(* IEC 61131-3 sources: AXOpen/src/components.rexroth.drives/ctrl/src/AxoCtrlxDriveXsc, 1 file *)

(* ---- AxoCtrlxDriveXsc.st ---- *)
USING AXOpen.Core;
USING AXOpen.Messaging.Static;
USING AXOpen.Messaging;
USING AXOpen.Core;
USING AXOpen.Components.Abstractions;
USING AXOpen.Components.Abstractions.Drives;
USING AXOpen.Components.Drives;
USING System.Math;
USING Siemens.Simatic.Hardware.Utilities;
USING Siemens.Simatic.DistributedIO;

NAMESPACE AXOpen.Components.Rexroth.Drives
    {S7.extern=ReadWrite}
    CLASS AxoCtrlxDriveXsc EXTENDS AXOpen.Components.Drives.AxoDrive IMPLEMENTS AXOpen.Components.Abstractions.Drives.IAxoDrive
        VAR PUBLIC //STATUS
            {#ix-attr:[Container(Layout.Stack)]}
            {#ix-attr:[ComponentDetails("Status")]}
            {#ix-attr:[ReadOnly()]}
            DriveStatus         :   AxoCtrlxDriveXsc_Component_Status;
            Messenger           :   AXOpen.Messaging.Static.AxoMessenger;
            TaskMessenger       :   AXOpen.Messaging.Static.AxoMessenger;
        END_VAR
        VAR PUBLIC // HwDiag
            {#ix-attr:[Container(Layout.Stack)]}
            {#ix-attr:[ComponentDetails("Hardware diagnostics")]}
            {#ix-set:AttributeName = "<#Update diagnostics#>"}
            HardwareDiagnosticsTask :   AXOpen.Io.AxoHardwareDiagnostics;
        END_VAR
        VAR PUBLIC // AxisRef
            {#ix-attr:[Container(Layout.Stack)]}
            {#ix-attr:[ComponentDetails("AxisRef")]}
            {#ix-attr:[ReadOnly()]}
            AxisRefExt :  AXOpen.Components.Rexroth.Drives.AxoCtrlxDriveXscAxisReference;
        END_VAR
        VAR PUBLIC // Scaling
            {#ix-attr:[Container(Layout.Stack)]}
            {#ix-attr:[ComponentDetails("Scaling")]}
            {#ix-attr:[ReadOnly()]}
            {#ix-set:AttributeName = "<#Scaling constant required position#>"}
            {#ix-set:AttributeToolTip = "<#Depends on the actual settings in the ctrlX DRIVE Engineering#>"}
            ScalingConstantRequiredPosition         :   LREAL   :=  10000.0;
            {#ix-attr:[ComponentDetails("Scaling")]}
            {#ix-attr:[ReadOnly()]}
            {#ix-set:AttributeName = "<#Scaling constant actual position#>"}
            {#ix-set:AttributeToolTip = "<#Depends on the actual settings in the ctrlX DRIVE Engineering#>"}
            ScalingConstantActualPosition         :   LREAL   :=  0.0001;
            {#ix-attr:[ComponentDetails("Scaling")]}
            {#ix-attr:[ReadOnly()]}
            {#ix-set:AttributeName = "<#Scaling constant required velocity#>"}
            {#ix-set:AttributeToolTip = "<#Depends on the actual settings in the ctrlX DRIVE Engineering#>"}
            ScalingConstantRequiredVelocity         :   LREAL   :=  LREAL#0.01666666666666666666666666666667;
            {#ix-attr:[ComponentDetails("Scaling")]}
            {#ix-attr:[ReadOnly()]}
            {#ix-set:AttributeName = "<#Scaling constant actual velocity#>"}
            {#ix-set:AttributeToolTip = "<#Depends on the actual settings in the ctrlX DRIVE Engineering#>"}
            ScalingConstantActualVelocity         :   LREAL   :=  60.0;
            {#ix-attr:[ComponentDetails("Scaling")]}
            {#ix-attr:[ReadOnly()]}
            {#ix-set:AttributeName = "<#Scaling constant required torque#>"}
            {#ix-set:AttributeToolTip = "<#Depends on the actual settings in the ctrlX DRIVE Engineering#>"}
            ScalingConstantRequiredTorque         :   LREAL   :=  10.0;
            {#ix-attr:[ComponentDetails("Scaling")]}
            {#ix-attr:[ReadOnly()]}
            {#ix-set:AttributeName = "<#Scaling constant actual torque#>"}
            {#ix-set:AttributeToolTip = "<#Depends on the actual settings in the ctrlX DRIVE Engineering#>"}
            ScalingConstantActualTorque         :   LREAL   :=  0.1;
            {#ix-attr:[ComponentDetails("Scaling")]}
            {#ix-attr:[ReadOnly()]}
            {#ix-set:AttributeName = "<#Scaling constant required acceleration#>"}
            {#ix-set:AttributeToolTip = "<#Depends on the actual settings in the ctrlX DRIVE Engineering#>"}
            ScalingConstantRequiredAcceleration        :   LREAL   :=  1000.0;
            {#ix-attr:[ComponentDetails("Scaling")]}
            {#ix-attr:[ReadOnly()]}
            {#ix-set:AttributeName = "<#Scaling constant actual acceleration#>"}
            {#ix-set:AttributeToolTip = "<#Depends on the actual settings in the ctrlX DRIVE Engineering#>"}
            ScalingConstantActualAcceleration        :   LREAL   :=  0.001;
            {#ix-attr:[ComponentDetails("Scaling")]}
            {#ix-attr:[ReadOnly()]}
            {#ix-set:AttributeName = "<#Scaling constant required deceleration#>"}
            {#ix-set:AttributeToolTip = "<#Depends on the actual settings in the ctrlX DRIVE Engineering#>"}
            ScalingConstantRequiredDeceleration        :   LREAL   :=  1000.0;
            {#ix-attr:[ComponentDetails("Scaling")]}
            {#ix-attr:[ReadOnly()]}
            {#ix-set:AttributeName = "<#Scaling constant actual deceleration#>"}
            {#ix-set:AttributeToolTip = "<#Depends on the actual settings in the ctrlX DRIVE Engineering#>"}
            ScalingConstantActualDeceleration        :   LREAL   :=  0.001;
            {#ix-set:AttributeName = "<#Scaling constant required jerk#>"}
            {#ix-set:AttributeToolTip = "<#Depends on the actual settings in the ctrlX DRIVE Engineering#>"}
            ScalingConstantRequiredJerk        :   LREAL   :=  1000.0;
            {#ix-attr:[ComponentDetails("Scaling")]}
            {#ix-attr:[ReadOnly()]}
            {#ix-set:AttributeName = "<#Scaling constant actual jerk#>"}
            {#ix-set:AttributeToolTip = "<#Depends on the actual settings in the ctrlX DRIVE Engineering#>"}
            ScalingConstantActualJerk       :   LREAL   :=  0.001;
            {#ix-attr:[ComponentDetails("Scaling")]}
            {#ix-attr:[ReadOnly()]}
            {#ix-set:AttributeName = "<#Axis type#>"}
            {#ix-set:AttributeToolTip = "<#Depends on the actual settings in the ctrlX DRIVE Engineering#>"}
            AxisType    :   eAxoDriveAxisType := eAxoDriveAxisType#Undefined;
        END_VAR
        VAR PUBLIC // Debug
            {#ix-attr:[Container(Layout.Stack)]}
            {#ix-attr:[ComponentHeader()]}
            {#ix-attr:[ReadOnly()]}
            {#ix-set:AttributeName = "<#_State#>"}
            _State                  :   UINT;
        END_VAR

        VAR PRIVATE
            _data2      :   ARRAY[0..1] OF BYTE;
            _data4      :   ARRAY[0..3] OF BYTE;
            _data8      :   ARRAY[0..7] OF BYTE;
            _word       :   WORD;
            _dword      :   DWORD;
            _lword      :   LWORD;

            _Parameter  : ARRAY[0..9] OF BYTE;
            _Fieldbus   : ARRAY[0..25] OF BYTE;

            _initHwCheckDone        :   BOOL;
            _retval                 :   WORD;
            _geoAddr                :   GeoAddr;
            _outHwid                :   UINT;
            _blink                  :   AXOpen.Timers.AxoBlinker;
            _inputsAddress          :   UDINT;
            _inputsCount            :   UINT;
            _outputsAddress         :   UDINT;
            _outputsCount           :   UINT;
            _ReadRecord             :   ReadRecord;
            _WriteRecord            :   WriteRecord;
            _ScalingRead            :   BOOL;
            _S_0_0076               :   WORD;       // 2byte, binary - Position data scaling type
            _S_0_0077               :   INT;        // 2byte, 0 decimal places - Linear position scaling factor
            _S_0_0078               :   INT;        // 2byte, 0 decimal places - Linear position scaling exponent
            _S_0_0079               :   DINT;       // 4byte, 0 decimal places - Rotational resolution
            _S_0_0044               :   WORD;       // 2byte, binary - Velocity scaling type
            _S_0_0045               :   INT;        // 2byte, 0 decimal places - Velocity scaling factor
            _S_0_0046               :   INT;        // 2byte, 0 decimal places - Velocity scaling exponent
            _S_0_0160               :   WORD;       // 2byte, binary - Acceleration scaling type
            _S_0_0161               :   INT;        // 2byte, 0 decimal places - Acceleration scaling factor
            _S_0_0162               :   INT;        // 2byte, 0 decimal places - Acceleration scaling exponent
            _S_0_0086               :   WORD;       // 2byte, binary - Torque/force scaling type
            _S_0_0093               :   INT;        // 2byte, 0 decimal places - Torque/force scaling factor
            _S_0_0094               :   INT;        // 2byte, 0 decimal places - Torque/force scaling exponent
            _S_0_0112               :   REAL;       // 4bytes, 3decimal places - Nominal current [A]
            _P_0_0450               :   REAL;       // 2bytes, 2decimal places - Current constant [Nm/A]

            _infoTimer              :   AXOpen.Timers.OnDelayTimer;
            _errorTimer             :   AXOpen.Timers.OnDelayTimer;
            _tmpTimer               :   AXOpen.Timers.OnDelayTimer;

            _lastMessageCodeFromMC  :   ULINT;
        END_VAR

        ///<summary>
        /// Runs tasks and logic of this component.
        /// >[!IMPORTANT] This method or one of its overloads must be called cyclically.
        ///</summary>
        METHOD PUBLIC Run
            VAR_INPUT
                inParent            :   IAxoObject;
                hwID                :   UINT;
                Enable              :   BOOL;                       //  As long as ‘Enable’ is true, power is being enabled.
                EnablePositive      :   BOOL;                       //  As long as ‘Enable’ is true, this permits motion in positive direction
                EnableNegative      :   BOOL;                       //  As long as ‘Enable’ is true, this permits motion in negative direction
            END_VAR
            VAR
                //                                      |     -10   |     -9    |    -8    |    -7   |   -6   |   -5  |  -4  | -3  | -2 |-1|  0 | 1  |  2  |  3   |   4   |   5    |   6     |    7     |     8     |    9      |     10    |
                _exp    :   ARRAY [-10..10] OF LREAL := [0.000000001,0.000000001,0.00000001,0.0000001,0.000001,0.00001,0.0001,0.001,0.01,0.1,1.0,10.0,100.0,1000.0,10000.0,100000.0,1000000.0,10000000.0,100000000.0,100000000.0,100000000.0];
            END_VAR
            SUPER.Run(inParent);
            Messenger.Serve(THIS);

            IF NOT _initHwCheckDone THEN
                IF inParent = NULL THEN
                    Messenger.Activate(     UINT#700, eAxoMessageCategory#ProgrammingError);
                    DriveStatus.Error.Id := UINT#700;
                    RETURN;
                END_IF;
                AxisRefExt.HWIDs.HW_Device :=  hwID;
                IF AxisRefExt.HWIDs.HW_Device = UINT#0 THEN
                    Messenger.Activate(     UINT#701, eAxoMessageCategory#ProgrammingError);
                    DriveStatus.Error.Id := UINT#701;
                    RETURN;
                END_IF;

                _retval := ReadSlotFromHardwareID(hardwareID := AxisRefExt.HWIDs.HW_Device, geoAddr :=_geoAddr);
                IF _retval = WORD#8090 THEN
                    Messenger.Activate(     UINT#702,eAxoMessageCategory#Error);
                    DriveStatus.Error.Id := UINT#702;
                    RETURN;
                END_IF;

                //******************Slot 1*****************//
                _geoAddr.Slot   :=  UINT#1;
                _geoAddr.HardwareType := UINT#4; // (4-Module)
                _retval := ReadHardwareIDFromSlot(geoAddr := _geoAddr, hardwareID => AxisRefExt.HWIDs.HW_Outputs);
                IF AxisRefExt.HWIDs.HW_Outputs = UINT#0 THEN
                    Messenger.Activate(     UINT#710,eAxoMessageCategory#Error);
                    DriveStatus.Error.Id := UINT#710;
                    RETURN;
                END_IF;
                IF _retval = WORD#8091 THEN
                    Messenger.Activate(     UINT#711,eAxoMessageCategory#Error);
                    DriveStatus.Error.Id := UINT#711;
                    RETURN;
                END_IF;
                IF _retval = WORD#8094 THEN
                    Messenger.Activate(     UINT#712,eAxoMessageCategory#Error);
                    DriveStatus.Error.Id := UINT#712;
                    RETURN;
                END_IF;
                IF _retval = WORD#8095 THEN
                    Messenger.Activate(     UINT#713,eAxoMessageCategory#Error);
                    DriveStatus.Error.Id := UINT#713;
                    RETURN;
                END_IF;
                IF _retval = WORD#8096 THEN
                    Messenger.Activate(     UINT#714,eAxoMessageCategory#Error);
                    DriveStatus.Error.Id := UINT#714;
                    RETURN;
                END_IF;
                IF _retval = WORD#8097 THEN
                    Messenger.Activate(     UINT#715,eAxoMessageCategory#Error);
                    DriveStatus.Error.Id := UINT#715;
                    RETURN;
                END_IF;
                ReadHardwareIOAddress(hardwareID := (AxisRefExt.HWIDs.HW_Outputs), inputStartAddress => _inputsAddress , inputCount => _inputsCount , outputStartAddress => _outputsAddress , outputCount => _outputsCount);
                IF _inputsCount <> UINT#0 OR _outputsCount <> UINT#0 THEN
                    Messenger.Activate(     UINT#716,eAxoMessageCategory#Error);
                    DriveStatus.Error.Id := UINT#716;
                    RETURN;
                END_IF;
                //******************Slot 2*****************//
                _geoAddr.Slot   :=  UINT#2;
                _geoAddr.HardwareType := UINT#4; // (4-Module)
                _retval := ReadHardwareIDFromSlot(geoAddr := _geoAddr, hardwareID =>  AxisRefExt.HWIDs.HW_Inputs);
                IF AxisRefExt.HWIDs.HW_Inputs = UINT#0 THEN
                    Messenger.Activate(     UINT#720,eAxoMessageCategory#Error);
                    DriveStatus.Error.Id := UINT#720;
                    RETURN;
                END_IF;
                IF _retval = WORD#8091 THEN
                    Messenger.Activate(     UINT#721,eAxoMessageCategory#Error);
                    DriveStatus.Error.Id := UINT#721;
                    RETURN;
                END_IF;
                IF _retval = WORD#8094 THEN
                    Messenger.Activate(     UINT#722,eAxoMessageCategory#Error);
                    DriveStatus.Error.Id := UINT#722;
                    RETURN;
                END_IF;
                IF _retval = WORD#8095 THEN
                    Messenger.Activate(     UINT#723,eAxoMessageCategory#Error);
                    DriveStatus.Error.Id := UINT#723;
                    RETURN;
                END_IF;
                IF _retval = WORD#8096 THEN
                    Messenger.Activate(     UINT#724,eAxoMessageCategory#Error);
                    DriveStatus.Error.Id := UINT#724;
                    RETURN;
                END_IF;
                IF _retval = WORD#8097 THEN
                    Messenger.Activate(     UINT#725,eAxoMessageCategory#Error);
                    DriveStatus.Error.Id := UINT#725;
                    RETURN;
                END_IF;
                ReadHardwareIOAddress(hardwareID := (AxisRefExt.HWIDs.HW_Inputs), inputStartAddress => _inputsAddress , inputCount => _inputsCount , outputStartAddress => _outputsAddress , outputCount => _outputsCount);
                IF _inputsCount <> UINT#0 OR _outputsCount <> UINT#0 THEN
                    Messenger.Activate(     UINT#726,eAxoMessageCategory#Error);
                    DriveStatus.Error.Id := UINT#726;
                    RETURN;
                END_IF;
                //************Slot 1 Subslot 1*****************//
                _geoAddr.Subslot:=      UINT#1;
                _geoAddr.Slot   :=      UINT#1;
                _geoAddr.HardwareType := UINT#5; // (5-Submodule)
                _retval := ReadHardwareIDFromSlot(geoAddr := _geoAddr, hardwareID => AxisRefExt.HWIDs.HW_S_0_0134_0_0);
                IF AxisRefExt.HWIDs.HW_S_0_0134_0_0  = UINT#0 THEN
                    Messenger.Activate(     UINT#730,eAxoMessageCategory#Error);
                    DriveStatus.Error.Id := UINT#730;
                    RETURN;
                END_IF;
                IF _retval = WORD#8091 THEN
                    Messenger.Activate(     UINT#731,eAxoMessageCategory#Error);
                    DriveStatus.Error.Id := UINT#731;
                    RETURN;
                END_IF;
                IF _retval = WORD#8094 THEN
                    Messenger.Activate(     UINT#732,eAxoMessageCategory#Error);
                    DriveStatus.Error.Id := UINT#732;
                    RETURN;
                END_IF;
                IF _retval = WORD#8095 THEN
                    Messenger.Activate(     UINT#733,eAxoMessageCategory#Error);
                    DriveStatus.Error.Id := UINT#733;
                    RETURN;
                END_IF;
                IF _retval = WORD#8096 THEN
                    Messenger.Activate(     UINT#734,eAxoMessageCategory#Error);
                    DriveStatus.Error.Id := UINT#734;
                    RETURN;
                END_IF;
                IF _retval = WORD#8097 THEN
                    Messenger.Activate(     UINT#735,eAxoMessageCategory#Error);
                    DriveStatus.Error.Id := UINT#735;
                    RETURN;
                END_IF;
                ReadHardwareIOAddress(hardwareID := (AxisRefExt.HWIDs.HW_S_0_0134_0_0) , inputStartAddress => _inputsAddress , inputCount => _inputsCount , outputStartAddress => _outputsAddress , outputCount => _outputsCount);
                IF _inputsCount <> UINT#0 OR _outputsCount <> UINT#2 THEN
                    Messenger.Activate(     UINT#736,eAxoMessageCategory#Error);
                    DriveStatus.Error.Id := UINT#736;
                    RETURN;
                END_IF;
                //************Slot 1 Subslot 2*****************//
                _geoAddr.Subslot:=      UINT#2;
                _geoAddr.Slot   :=      UINT#1;
                _geoAddr.HardwareType := UINT#5; // (5-Submodule)
                _retval := ReadHardwareIDFromSlot(geoAddr := _geoAddr, hardwareID => AxisRefExt.HWIDs.HW_S_0_0145_0_0);
                IF AxisRefExt.HWIDs.HW_S_0_0145_0_0  = UINT#0 THEN
                    Messenger.Activate(     UINT#740,eAxoMessageCategory#Error);
                    DriveStatus.Error.Id := UINT#740;
                    RETURN;
                END_IF;
                IF _retval = WORD#8091 THEN
                    Messenger.Activate(     UINT#741,eAxoMessageCategory#Error);
                    DriveStatus.Error.Id := UINT#741;
                    RETURN;
                END_IF;
                IF _retval = WORD#8094 THEN
                    Messenger.Activate(     UINT#742,eAxoMessageCategory#Error);
                    DriveStatus.Error.Id := UINT#742;
                    RETURN;
                END_IF;
                IF _retval = WORD#8095 THEN
                    Messenger.Activate(     UINT#743,eAxoMessageCategory#Error);
                    DriveStatus.Error.Id := UINT#743;
                    RETURN;
                END_IF;
                IF _retval = WORD#8096 THEN
                    Messenger.Activate(     UINT#744,eAxoMessageCategory#Error);
                    DriveStatus.Error.Id := UINT#744;
                    RETURN;
                END_IF;
                IF _retval = WORD#8097 THEN
                    Messenger.Activate(     UINT#745,eAxoMessageCategory#Error);
                    DriveStatus.Error.Id := UINT#745;
                    RETURN;
                END_IF;
                ReadHardwareIOAddress(hardwareID := (AxisRefExt.HWIDs.HW_S_0_0145_0_0) , inputStartAddress => _inputsAddress , inputCount => _inputsCount , outputStartAddress => _outputsAddress , outputCount => _outputsCount);
                IF _inputsCount <> UINT#0 OR _outputsCount <> UINT#2 THEN
                    Messenger.Activate(     UINT#746,eAxoMessageCategory#Error);
                    DriveStatus.Error.Id := UINT#746;
                    RETURN;
                END_IF;
                //************Slot 1 Subslot 3*****************//
                _geoAddr.Subslot:=      UINT#3;
                _geoAddr.Slot   :=      UINT#1;
                _geoAddr.HardwareType := UINT#5; // (5-Submodule)
                _retval := ReadHardwareIDFromSlot(geoAddr := _geoAddr, hardwareID => AxisRefExt.HWIDs.HW_S_0_0282_0_0);
                IF AxisRefExt.HWIDs.HW_S_0_0282_0_0  = UINT#0 THEN
                    Messenger.Activate(     UINT#750,eAxoMessageCategory#Error);
                    DriveStatus.Error.Id := UINT#750;
                    RETURN;
                END_IF;
                IF _retval = WORD#8091 THEN
                    Messenger.Activate(     UINT#751,eAxoMessageCategory#Error);
                    DriveStatus.Error.Id := UINT#751;
                    RETURN;
                END_IF;
                IF _retval = WORD#8094 THEN
                    Messenger.Activate(     UINT#752,eAxoMessageCategory#Error);
                    DriveStatus.Error.Id := UINT#752;
                    RETURN;
                END_IF;
                IF _retval = WORD#8095 THEN
                    Messenger.Activate(     UINT#753,eAxoMessageCategory#Error);
                    DriveStatus.Error.Id := UINT#753;
                    RETURN;
                END_IF;
                IF _retval = WORD#8096 THEN
                    Messenger.Activate(     UINT#754,eAxoMessageCategory#Error);
                    DriveStatus.Error.Id := UINT#754;
                    RETURN;
                END_IF;
                IF _retval = WORD#8097 THEN
                    Messenger.Activate(     UINT#755,eAxoMessageCategory#Error);
                    DriveStatus.Error.Id := UINT#755;
                    RETURN;
                END_IF;
                ReadHardwareIOAddress(hardwareID := (AxisRefExt.HWIDs.HW_S_0_0282_0_0) , inputStartAddress => _inputsAddress , inputCount => _inputsCount , outputStartAddress => _outputsAddress , outputCount => _outputsCount);
                IF _inputsCount <> UINT#0 OR _outputsCount <> UINT#4 THEN
                    Messenger.Activate(     UINT#756,eAxoMessageCategory#Error);
                    DriveStatus.Error.Id := UINT#756;
                    RETURN;
                END_IF;
                //************Slot 1 Subslot 4*****************//
                _geoAddr.Subslot:=      UINT#4;
                _geoAddr.Slot   :=      UINT#1;
                _geoAddr.HardwareType := UINT#5; // (5-Submodule)
                _retval := ReadHardwareIDFromSlot(geoAddr := _geoAddr, hardwareID => AxisRefExt.HWIDs.HW_S_0_0259_0_0);
                IF AxisRefExt.HWIDs.HW_S_0_0259_0_0  = UINT#0 THEN
                    Messenger.Activate(     UINT#760,eAxoMessageCategory#Error);
                    DriveStatus.Error.Id := UINT#760;
                    RETURN;
                END_IF;
                IF _retval = WORD#8091 THEN
                    Messenger.Activate(     UINT#761,eAxoMessageCategory#Error);
                    DriveStatus.Error.Id := UINT#761;
                    RETURN;
                END_IF;
                IF _retval = WORD#8094 THEN
                    Messenger.Activate(     UINT#762,eAxoMessageCategory#Error);
                    DriveStatus.Error.Id := UINT#762;
                    RETURN;
                END_IF;
                IF _retval = WORD#8095 THEN
                    Messenger.Activate(     UINT#763,eAxoMessageCategory#Error);
                    DriveStatus.Error.Id := UINT#763;
                    RETURN;
                END_IF;
                IF _retval = WORD#8096 THEN
                    Messenger.Activate(     UINT#764,eAxoMessageCategory#Error);
                    DriveStatus.Error.Id := UINT#764;
                    RETURN;
                END_IF;
                IF _retval = WORD#8097 THEN
                    Messenger.Activate(     UINT#765,eAxoMessageCategory#Error);
                    DriveStatus.Error.Id := UINT#765;
                    RETURN;
                END_IF;
                ReadHardwareIOAddress(hardwareID := (AxisRefExt.HWIDs.HW_S_0_0259_0_0) , inputStartAddress => _inputsAddress , inputCount => _inputsCount , outputStartAddress => _outputsAddress , outputCount => _outputsCount);
                IF _inputsCount <> UINT#0 OR _outputsCount <> UINT#4 THEN
                    Messenger.Activate(     UINT#766,eAxoMessageCategory#Error);
                    DriveStatus.Error.Id := UINT#766;
                    RETURN;
                END_IF;
                //************Slot 1 Subslot 5*****************//
                _geoAddr.Subslot:=      UINT#5;
                _geoAddr.Slot   :=      UINT#1;
                _geoAddr.HardwareType := UINT#5; // (5-Submodule)
                _retval := ReadHardwareIDFromSlot(geoAddr := _geoAddr, hardwareID => AxisRefExt.HWIDs.HW_S_0_0260_0_0);
                IF AxisRefExt.HWIDs.HW_S_0_0260_0_0  = UINT#0 THEN
                    Messenger.Activate(     UINT#770,eAxoMessageCategory#Error);
                    DriveStatus.Error.Id := UINT#770;
                    RETURN;
                END_IF;
                IF _retval = WORD#8091 THEN
                    Messenger.Activate(     UINT#771,eAxoMessageCategory#Error);
                    DriveStatus.Error.Id := UINT#771;
                    RETURN;
                END_IF;
                IF _retval = WORD#8094 THEN
                    Messenger.Activate(     UINT#772,eAxoMessageCategory#Error);
                    DriveStatus.Error.Id := UINT#772;
                    RETURN;
                END_IF;
                IF _retval = WORD#8095 THEN
                    Messenger.Activate(     UINT#773,eAxoMessageCategory#Error);
                    DriveStatus.Error.Id := UINT#773;
                    RETURN;
                END_IF;
                IF _retval = WORD#8096 THEN
                    Messenger.Activate(     UINT#774,eAxoMessageCategory#Error);
                    DriveStatus.Error.Id := UINT#774;
                    RETURN;
                END_IF;
                IF _retval = WORD#8097 THEN
                    Messenger.Activate(     UINT#775,eAxoMessageCategory#Error);
                    DriveStatus.Error.Id := UINT#775;
                    RETURN;
                END_IF;
                ReadHardwareIOAddress(hardwareID := (AxisRefExt.HWIDs.HW_S_0_0260_0_0) , inputStartAddress => _inputsAddress , inputCount => _inputsCount , outputStartAddress => _outputsAddress , outputCount => _outputsCount);
                IF _inputsCount <> UINT#0 OR _outputsCount <> UINT#4 THEN
                    Messenger.Activate(     UINT#776,eAxoMessageCategory#Error);
                    DriveStatus.Error.Id := UINT#776;
                    RETURN;
                END_IF;
                //************Slot 1 Subslot 6*****************//
                _geoAddr.Subslot:=      UINT#6;
                _geoAddr.Slot   :=      UINT#1;
                _geoAddr.HardwareType := UINT#5; // (5-Submodule)
                _retval := ReadHardwareIDFromSlot(geoAddr := _geoAddr, hardwareID => AxisRefExt.HWIDs.HW_S_0_0359_0_0);
                IF AxisRefExt.HWIDs.HW_S_0_0359_0_0 = UINT#0 THEN
                    Messenger.Activate(     UINT#780,eAxoMessageCategory#Error);
                    DriveStatus.Error.Id := UINT#780;
                    RETURN;
                END_IF;
                IF _retval = WORD#8091 THEN
                    Messenger.Activate(     UINT#781,eAxoMessageCategory#Error);
                    DriveStatus.Error.Id := UINT#781;
                    RETURN;
                END_IF;
                IF _retval = WORD#8094 THEN
                    Messenger.Activate(     UINT#782,eAxoMessageCategory#Error);
                    DriveStatus.Error.Id := UINT#782;
                    RETURN;
                END_IF;
                IF _retval = WORD#8095 THEN
                    Messenger.Activate(     UINT#783,eAxoMessageCategory#Error);
                    DriveStatus.Error.Id := UINT#783;
                    RETURN;
                END_IF;
                IF _retval = WORD#8096 THEN
                    Messenger.Activate(     UINT#784,eAxoMessageCategory#Error);
                    DriveStatus.Error.Id := UINT#784;
                    RETURN;
                END_IF;
                IF _retval = WORD#8097 THEN
                    Messenger.Activate(     UINT#785,eAxoMessageCategory#Error);
                    DriveStatus.Error.Id := UINT#785;
                    RETURN;
                END_IF;
                ReadHardwareIOAddress(hardwareID := (AxisRefExt.HWIDs.HW_S_0_0359_0_0) , inputStartAddress => _inputsAddress , inputCount => _inputsCount , outputStartAddress => _outputsAddress , outputCount => _outputsCount);
                IF _inputsCount <> UINT#0 OR _outputsCount <> UINT#4 THEN
                    Messenger.Activate(     UINT#786,eAxoMessageCategory#Error);
                    DriveStatus.Error.Id := UINT#786;
                    RETURN;
                END_IF;
                //************Slot 1 Subslot 7*****************//
                _geoAddr.Subslot:=      UINT#7;
                _geoAddr.Slot   :=      UINT#1;
                _geoAddr.HardwareType := UINT#5; // (5-Submodule)
                _retval := ReadHardwareIDFromSlot(geoAddr := _geoAddr, hardwareID => AxisRefExt.HWIDs.HW_S_0_1720_0_1);
                IF AxisRefExt.HWIDs.HW_S_0_1720_0_1 = UINT#0 THEN
                    Messenger.Activate(     UINT#790,eAxoMessageCategory#Error);
                    DriveStatus.Error.Id := UINT#790;
                    RETURN;
                END_IF;
                IF _retval = WORD#8091 THEN
                    Messenger.Activate(     UINT#791,eAxoMessageCategory#Error);
                    DriveStatus.Error.Id := UINT#791;
                    RETURN;
                END_IF;
                IF _retval = WORD#8094 THEN
                    Messenger.Activate(     UINT#792,eAxoMessageCategory#Error);
                    DriveStatus.Error.Id := UINT#792;
                    RETURN;
                END_IF;
                IF _retval = WORD#8095 THEN
                    Messenger.Activate(     UINT#793,eAxoMessageCategory#Error);
                    DriveStatus.Error.Id := UINT#793;
                    RETURN;
                END_IF;
                IF _retval = WORD#8096 THEN
                    Messenger.Activate(     UINT#794,eAxoMessageCategory#Error);
                    DriveStatus.Error.Id := UINT#794;
                    RETURN;
                END_IF;
                IF _retval = WORD#8097 THEN
                    Messenger.Activate(     UINT#795,eAxoMessageCategory#Error);
                    DriveStatus.Error.Id := UINT#795;
                    RETURN;
                END_IF;
                ReadHardwareIOAddress(hardwareID := (AxisRefExt.HWIDs.HW_S_0_1720_0_1) , inputStartAddress => _inputsAddress , inputCount => _inputsCount , outputStartAddress => _outputsAddress , outputCount => _outputsCount);
                IF _inputsCount <> UINT#0 OR _outputsCount <> UINT#2 THEN
                    Messenger.Activate(     UINT#796,eAxoMessageCategory#Error);
                    DriveStatus.Error.Id := UINT#796;
                    RETURN;
                END_IF;
                //************Slot 1 Subslot 8*****************//
                _geoAddr.Subslot:=      UINT#8;
                _geoAddr.Slot   :=      UINT#1;
                _geoAddr.HardwareType := UINT#5; // (5-Submodule)
                _retval := ReadHardwareIDFromSlot(geoAddr := _geoAddr, hardwareID => AxisRefExt.HWIDs.HW_S_0_0092_0_0);
                IF AxisRefExt.HWIDs.HW_S_0_0092_0_0  = UINT#0 THEN
                    Messenger.Activate(     UINT#800,eAxoMessageCategory#Error);
                    DriveStatus.Error.Id := UINT#800;
                    RETURN;
                END_IF;
                IF _retval = WORD#8091 THEN
                    Messenger.Activate(     UINT#801,eAxoMessageCategory#Error);
                    DriveStatus.Error.Id := UINT#801;
                    RETURN;
                END_IF;
                IF _retval = WORD#8094 THEN
                    Messenger.Activate(     UINT#802,eAxoMessageCategory#Error);
                    DriveStatus.Error.Id := UINT#802;
                    RETURN;
                END_IF;
                IF _retval = WORD#8095 THEN
                    Messenger.Activate(     UINT#803,eAxoMessageCategory#Error);
                    DriveStatus.Error.Id := UINT#803;
                    RETURN;
                END_IF;
                IF _retval = WORD#8096 THEN
                    Messenger.Activate(     UINT#804,eAxoMessageCategory#Error);
                    DriveStatus.Error.Id := UINT#804;
                    RETURN;
                END_IF;
                IF _retval = WORD#8097 THEN
                    Messenger.Activate(     UINT#805,eAxoMessageCategory#Error);
                    DriveStatus.Error.Id := UINT#805;
                    RETURN;
                END_IF;
                ReadHardwareIOAddress(hardwareID := (AxisRefExt.HWIDs.HW_S_0_0092_0_0) , inputStartAddress => _inputsAddress , inputCount => _inputsCount , outputStartAddress => _outputsAddress , outputCount => _outputsCount);
                IF _inputsCount <> UINT#0 OR _outputsCount <> UINT#2 THEN
                    Messenger.Activate(     UINT#806,eAxoMessageCategory#Error);
                    DriveStatus.Error.Id := UINT#806;
                    RETURN;
                END_IF;
                //************Slot 1 Subslot 9*****************//
                _geoAddr.Subslot:=      UINT#9;
                _geoAddr.Slot   :=      UINT#1;
                _geoAddr.HardwareType := UINT#5; // (5-Submodule)
                _retval := ReadHardwareIDFromSlot(geoAddr := _geoAddr, hardwareID => AxisRefExt.HWIDs.HW_S_0_0080_0_0);
                IF AxisRefExt.HWIDs.HW_S_0_0080_0_0  = UINT#0 THEN
                    Messenger.Activate(     UINT#810,eAxoMessageCategory#Error);
                    DriveStatus.Error.Id := UINT#810;
                    RETURN;
                END_IF;
                IF _retval = WORD#8091 THEN
                    Messenger.Activate(     UINT#811,eAxoMessageCategory#Error);
                    DriveStatus.Error.Id := UINT#811;
                    RETURN;
                END_IF;
                IF _retval = WORD#8094 THEN
                    Messenger.Activate(     UINT#812,eAxoMessageCategory#Error);
                    DriveStatus.Error.Id := UINT#812;
                    RETURN;
                END_IF;
                IF _retval = WORD#8095 THEN
                    Messenger.Activate(     UINT#813,eAxoMessageCategory#Error);
                    DriveStatus.Error.Id := UINT#813;
                    RETURN;
                END_IF;
                IF _retval = WORD#8096 THEN
                    Messenger.Activate(     UINT#814,eAxoMessageCategory#Error);
                    DriveStatus.Error.Id := UINT#814;
                    RETURN;
                END_IF;
                IF _retval = WORD#8097 THEN
                    Messenger.Activate(     UINT#815,eAxoMessageCategory#Error);
                    DriveStatus.Error.Id := UINT#815;
                    RETURN;
                END_IF;
                ReadHardwareIOAddress(hardwareID := (AxisRefExt.HWIDs.HW_S_0_0080_0_0) , inputStartAddress => _inputsAddress , inputCount => _inputsCount , outputStartAddress => _outputsAddress , outputCount => _outputsCount);
                IF _inputsCount <> UINT#0 OR _outputsCount <> UINT#2 THEN
                    Messenger.Activate(     UINT#816,eAxoMessageCategory#Error);
                    DriveStatus.Error.Id := UINT#816;
                    RETURN;
                END_IF;
                //************Slot 1 Subslot 10*****************//
                _geoAddr.Subslot:=      UINT#10;
                _geoAddr.Slot   :=      UINT#1;
                _geoAddr.HardwareType := UINT#5; // (5-Submodule)
                _retval := ReadHardwareIDFromSlot(geoAddr := _geoAddr, hardwareID =>  AxisRefExt.HWIDs.HW_S_0_0193_0_0);
                IF AxisRefExt.HWIDs.HW_S_0_0193_0_0 = UINT#0 THEN
                    Messenger.Activate(     UINT#820,eAxoMessageCategory#Error);
                    DriveStatus.Error.Id := UINT#820;
                    RETURN;
                END_IF;
                IF _retval = WORD#8091 THEN
                    Messenger.Activate(     UINT#821,eAxoMessageCategory#Error);
                    DriveStatus.Error.Id := UINT#821;
                    RETURN;
                END_IF;
                IF _retval = WORD#8094 THEN
                    Messenger.Activate(     UINT#822,eAxoMessageCategory#Error);
                    DriveStatus.Error.Id := UINT#822;
                    RETURN;
                END_IF;
                IF _retval = WORD#8095 THEN
                    Messenger.Activate(     UINT#823,eAxoMessageCategory#Error);
                    DriveStatus.Error.Id := UINT#823;
                    RETURN;
                END_IF;
                IF _retval = WORD#8096 THEN
                    Messenger.Activate(     UINT#824,eAxoMessageCategory#Error);
                    DriveStatus.Error.Id := UINT#824;
                    RETURN;
                END_IF;
                IF _retval = WORD#8097 THEN
                    Messenger.Activate(     UINT#825,eAxoMessageCategory#Error);
                    DriveStatus.Error.Id := UINT#825;
                    RETURN;
                END_IF;
                ReadHardwareIOAddress(hardwareID := (AxisRefExt.HWIDs.HW_S_0_0193_0_0) , inputStartAddress => _inputsAddress , inputCount => _inputsCount , outputStartAddress => _outputsAddress , outputCount => _outputsCount);
                IF _inputsCount <> UINT#0 OR _outputsCount <> UINT#4 THEN
                    Messenger.Activate(     UINT#826,eAxoMessageCategory#Error);
                    DriveStatus.Error.Id := UINT#826;
                    RETURN;
                END_IF;
                //************Slot 2 Subslot 1*****************//
                _geoAddr.Subslot:=      UINT#1;
                _geoAddr.Slot   :=      UINT#2;
                _geoAddr.HardwareType := UINT#5; // (5-Submodule)
                _retval := ReadHardwareIDFromSlot(geoAddr := _geoAddr, hardwareID => AxisRefExt.HWIDs.HW_S_0_0135_0_0);
                IF AxisRefExt.HWIDs.HW_S_0_0135_0_0  = UINT#0 THEN
                    Messenger.Activate(     UINT#830,eAxoMessageCategory#Error);
                    DriveStatus.Error.Id := UINT#830;
                    RETURN;
                END_IF;
                IF _retval = WORD#8091 THEN
                    Messenger.Activate(     UINT#831,eAxoMessageCategory#Error);
                    DriveStatus.Error.Id := UINT#831;
                    RETURN;
                END_IF;
                IF _retval = WORD#8094 THEN
                    Messenger.Activate(     UINT#832,eAxoMessageCategory#Error);
                    DriveStatus.Error.Id := UINT#832;
                    RETURN;
                END_IF;
                IF _retval = WORD#8095 THEN
                    Messenger.Activate(     UINT#833,eAxoMessageCategory#Error);
                    DriveStatus.Error.Id := UINT#833;
                    RETURN;
                END_IF;
                IF _retval = WORD#8096 THEN
                    Messenger.Activate(     UINT#834,eAxoMessageCategory#Error);
                    DriveStatus.Error.Id := UINT#834;
                    RETURN;
                END_IF;
                IF _retval = WORD#8097 THEN
                    Messenger.Activate(     UINT#835,eAxoMessageCategory#Error);
                    DriveStatus.Error.Id := UINT#835;
                    RETURN;
                END_IF;
                ReadHardwareIOAddress(hardwareID := (AxisRefExt.HWIDs.HW_S_0_0135_0_0) , inputStartAddress => _inputsAddress , inputCount => _inputsCount , outputStartAddress => _outputsAddress , outputCount => _outputsCount);
                IF _inputsCount <> UINT#2 OR _outputsCount <> UINT#0 THEN
                    Messenger.Activate(     UINT#836,eAxoMessageCategory#Error);
                    DriveStatus.Error.Id := UINT#836;
                    RETURN;
                END_IF;
                //************Slot 2 Subslot 2*****************//
                _geoAddr.Subslot:=      UINT#2;
                _geoAddr.Slot   :=      UINT#2;
                _geoAddr.HardwareType := UINT#5; // (5-Submodule)
                _retval := ReadHardwareIDFromSlot(geoAddr := _geoAddr, hardwareID => AxisRefExt.HWIDs.HW_S_0_0144_0_0);
                IF AxisRefExt.HWIDs.HW_S_0_0144_0_0  = UINT#0 THEN
                    Messenger.Activate(     UINT#840,eAxoMessageCategory#Error);
                    DriveStatus.Error.Id := UINT#840;
                    RETURN;
                END_IF;
                IF _retval = WORD#8091 THEN
                    Messenger.Activate(     UINT#841,eAxoMessageCategory#Error);
                    DriveStatus.Error.Id := UINT#841;
                    RETURN;
                END_IF;
                IF _retval = WORD#8094 THEN
                    Messenger.Activate(     UINT#842,eAxoMessageCategory#Error);
                    DriveStatus.Error.Id := UINT#842;
                    RETURN;
                END_IF;
                IF _retval = WORD#8095 THEN
                    Messenger.Activate(     UINT#843,eAxoMessageCategory#Error);
                    DriveStatus.Error.Id := UINT#843;
                    RETURN;
                END_IF;
                IF _retval = WORD#8096 THEN
                    Messenger.Activate(     UINT#844,eAxoMessageCategory#Error);
                    DriveStatus.Error.Id := UINT#844;
                    RETURN;
                END_IF;
                IF _retval = WORD#8097 THEN
                    Messenger.Activate(     UINT#845,eAxoMessageCategory#Error);
                    DriveStatus.Error.Id := UINT#845;
                    RETURN;
                END_IF;
                ReadHardwareIOAddress(hardwareID := (AxisRefExt.HWIDs.HW_S_0_0144_0_0) , inputStartAddress => _inputsAddress , inputCount => _inputsCount , outputStartAddress => _outputsAddress , outputCount => _outputsCount);
                IF _inputsCount <> UINT#2 OR _outputsCount <> UINT#0 THEN
                    Messenger.Activate(     UINT#846,eAxoMessageCategory#Error);
                    DriveStatus.Error.Id := UINT#846;
                    RETURN;
                END_IF;
                //************Slot 2 Subslot 3*****************//
                _geoAddr.Subslot:=      UINT#3;
                _geoAddr.Slot   :=      UINT#2;
                _geoAddr.HardwareType := UINT#5; // (5-Submodule)
                _retval := ReadHardwareIDFromSlot(geoAddr := _geoAddr, hardwareID => AxisRefExt.HWIDs.HW_S_0_0386_0_0);
                IF AxisRefExt.HWIDs.HW_S_0_0386_0_0 = UINT#0 THEN
                    Messenger.Activate(     UINT#850,eAxoMessageCategory#Error);
                    DriveStatus.Error.Id := UINT#850;
                    RETURN;
                END_IF;
                IF _retval = WORD#8091 THEN
                    Messenger.Activate(     UINT#851,eAxoMessageCategory#Error);
                    DriveStatus.Error.Id := UINT#851;
                    RETURN;
                END_IF;
                IF _retval = WORD#8094 THEN
                    Messenger.Activate(     UINT#852,eAxoMessageCategory#Error);
                    DriveStatus.Error.Id := UINT#852;
                    RETURN;
                END_IF;
                IF _retval = WORD#8095 THEN
                    Messenger.Activate(     UINT#853,eAxoMessageCategory#Error);
                    DriveStatus.Error.Id := UINT#853;
                    RETURN;
                END_IF;
                IF _retval = WORD#8096 THEN
                    Messenger.Activate(     UINT#854,eAxoMessageCategory#Error);
                    DriveStatus.Error.Id := UINT#854;
                    RETURN;
                END_IF;
                IF _retval = WORD#8097 THEN
                    Messenger.Activate(     UINT#855,eAxoMessageCategory#Error);
                    DriveStatus.Error.Id := UINT#855;
                    RETURN;
                END_IF;
                ReadHardwareIOAddress(hardwareID := (AxisRefExt.HWIDs.HW_S_0_0386_0_0) , inputStartAddress => _inputsAddress , inputCount => _inputsCount , outputStartAddress => _outputsAddress , outputCount => _outputsCount);
                IF _inputsCount <> UINT#4 OR _outputsCount <> UINT#0 THEN
                    Messenger.Activate(     UINT#856,eAxoMessageCategory#Error);
                    DriveStatus.Error.Id := UINT#856;
                    RETURN;
                END_IF;
                //************Slot 2 Subslot 4*****************//
                _geoAddr.Subslot:=      UINT#4;
                _geoAddr.Slot   :=      UINT#2;
                _geoAddr.HardwareType := UINT#5; // (5-Submodule)
                _retval := ReadHardwareIDFromSlot(geoAddr := _geoAddr, hardwareID => AxisRefExt.HWIDs.HW_S_0_0535_0_0);
                IF AxisRefExt.HWIDs.HW_S_0_0535_0_0  = UINT#0 THEN
                    Messenger.Activate(     UINT#860,eAxoMessageCategory#Error);
                    DriveStatus.Error.Id := UINT#860;
                    RETURN;
                END_IF;
                IF _retval = WORD#8091 THEN
                    Messenger.Activate(     UINT#861,eAxoMessageCategory#Error);
                    DriveStatus.Error.Id := UINT#861;
                    RETURN;
                END_IF;
                IF _retval = WORD#8094 THEN
                    Messenger.Activate(     UINT#862,eAxoMessageCategory#Error);
                    DriveStatus.Error.Id := UINT#862;
                    RETURN;
                END_IF;
                IF _retval = WORD#8095 THEN
                    Messenger.Activate(     UINT#863,eAxoMessageCategory#Error);
                    DriveStatus.Error.Id := UINT#863;
                    RETURN;
                END_IF;
                IF _retval = WORD#8096 THEN
                    Messenger.Activate(     UINT#864,eAxoMessageCategory#Error);
                    DriveStatus.Error.Id := UINT#864;
                    RETURN;
                END_IF;
                IF _retval = WORD#8097 THEN
                    Messenger.Activate(     UINT#865,eAxoMessageCategory#Error);
                    DriveStatus.Error.Id := UINT#865;
                    RETURN;
                END_IF;
                ReadHardwareIOAddress(hardwareID := (AxisRefExt.HWIDs.HW_S_0_0535_0_0) , inputStartAddress => _inputsAddress , inputCount => _inputsCount , outputStartAddress => _outputsAddress , outputCount => _outputsCount);
                IF _inputsCount <> UINT#4 OR _outputsCount <> UINT#0 THEN
                    Messenger.Activate(     UINT#866,eAxoMessageCategory#Error);
                    DriveStatus.Error.Id := UINT#866;
                    RETURN;
                END_IF;
                //************Slot 2 Subslot 5*****************//
                _geoAddr.Subslot:=      UINT#5;
                _geoAddr.Slot   :=      UINT#2;
                _geoAddr.HardwareType := UINT#5; // (5-Submodule)
                _retval := ReadHardwareIDFromSlot(geoAddr := _geoAddr, hardwareID => AxisRefExt.HWIDs.HW_S_0_0390_0_0);
                IF AxisRefExt.HWIDs.HW_S_0_0390_0_0  = UINT#0 THEN
                    Messenger.Activate(     UINT#870,eAxoMessageCategory#Error);
                    DriveStatus.Error.Id := UINT#870;
                    RETURN;
                END_IF;
                IF _retval = WORD#8091 THEN
                    Messenger.Activate(     UINT#871,eAxoMessageCategory#Error);
                    DriveStatus.Error.Id := UINT#871;
                    RETURN;
                END_IF;
                IF _retval = WORD#8094 THEN
                    Messenger.Activate(     UINT#872,eAxoMessageCategory#Error);
                    DriveStatus.Error.Id := UINT#872;
                    RETURN;
                END_IF;
                IF _retval = WORD#8095 THEN
                    Messenger.Activate(     UINT#873,eAxoMessageCategory#Error);
                    DriveStatus.Error.Id := UINT#873;
                    RETURN;
                END_IF;
                IF _retval = WORD#8096 THEN
                    Messenger.Activate(     UINT#874,eAxoMessageCategory#Error);
                    DriveStatus.Error.Id := UINT#874;
                    RETURN;
                END_IF;
                IF _retval = WORD#8097 THEN
                    Messenger.Activate(     UINT#875,eAxoMessageCategory#Error);
                    DriveStatus.Error.Id := UINT#875;
                    RETURN;
                END_IF;
                ReadHardwareIOAddress(hardwareID := (AxisRefExt.HWIDs.HW_S_0_0390_0_0), inputStartAddress => _inputsAddress , inputCount => _inputsCount , outputStartAddress => _outputsAddress , outputCount => _outputsCount);
                IF _inputsCount <> UINT#4 OR _outputsCount <> UINT#0 THEN
                    Messenger.Activate(     UINT#876,eAxoMessageCategory#Error);
                    DriveStatus.Error.Id := UINT#876;
                    RETURN;
                END_IF;
                //************Slot 2 Subslot 6*****************//
                _geoAddr.Subslot:=      UINT#6;
                _geoAddr.Slot   :=      UINT#2;
                _geoAddr.HardwareType := UINT#5; // (5-Submodule)
                _retval := ReadHardwareIDFromSlot(geoAddr := _geoAddr, hardwareID => AxisRefExt.HWIDs.HW_S_0_1720_0_2);
                IF AxisRefExt.HWIDs.HW_S_0_1720_0_2  = UINT#0 THEN
                    Messenger.Activate(     UINT#880,eAxoMessageCategory#Error);
                    DriveStatus.Error.Id := UINT#880;
                    RETURN;
                END_IF;
                IF _retval = WORD#8091 THEN
                    Messenger.Activate(     UINT#881,eAxoMessageCategory#Error);
                    DriveStatus.Error.Id := UINT#881;
                    RETURN;
                END_IF;
                IF _retval = WORD#8094 THEN
                    Messenger.Activate(     UINT#882,eAxoMessageCategory#Error);
                    DriveStatus.Error.Id := UINT#882;
                    RETURN;
                END_IF;
                IF _retval = WORD#8095 THEN
                    Messenger.Activate(     UINT#883,eAxoMessageCategory#Error);
                    DriveStatus.Error.Id := UINT#883;
                    RETURN;
                END_IF;
                IF _retval = WORD#8096 THEN
                    Messenger.Activate(     UINT#884,eAxoMessageCategory#Error);
                    DriveStatus.Error.Id := UINT#884;
                    RETURN;
                END_IF;
                IF _retval = WORD#8097 THEN
                    Messenger.Activate(     UINT#885,eAxoMessageCategory#Error);
                    DriveStatus.Error.Id := UINT#885;
                    RETURN;
                END_IF;
                ReadHardwareIOAddress(hardwareID := (AxisRefExt.HWIDs.HW_S_0_1720_0_2) , inputStartAddress => _inputsAddress , inputCount => _inputsCount , outputStartAddress => _outputsAddress , outputCount => _outputsCount);
                IF _inputsCount <> UINT#2 OR _outputsCount <> UINT#0 THEN
                    Messenger.Activate(     UINT#886,eAxoMessageCategory#Error);
                    DriveStatus.Error.Id := UINT#886;
                    RETURN;
                END_IF;
                //************Slot 2 Subslot 7*****************//
                _geoAddr.Subslot:=      UINT#7;
                _geoAddr.Slot   :=      UINT#2;
                _geoAddr.HardwareType := UINT#5; // (5-Submodule)
                _retval := ReadHardwareIDFromSlot(geoAddr := _geoAddr, hardwareID => AxisRefExt.HWIDs.HW_S_0_0084_0_0);
                IF AxisRefExt.HWIDs.HW_S_0_0084_0_0  = UINT#0 THEN
                    Messenger.Activate(     UINT#890,eAxoMessageCategory#Error);
                    DriveStatus.Error.Id := UINT#890;
                    RETURN;
                END_IF;
                IF _retval = WORD#8091 THEN
                    Messenger.Activate(     UINT#891,eAxoMessageCategory#Error);
                    DriveStatus.Error.Id := UINT#891;
                    RETURN;
                END_IF;
                IF _retval = WORD#8094 THEN
                    Messenger.Activate(     UINT#892,eAxoMessageCategory#Error);
                    DriveStatus.Error.Id := UINT#892;
                    RETURN;
                END_IF;
                IF _retval = WORD#8095 THEN
                    Messenger.Activate(     UINT#893,eAxoMessageCategory#Error);
                    DriveStatus.Error.Id := UINT#893;
                    RETURN;
                END_IF;
                IF _retval = WORD#8096 THEN
                    Messenger.Activate(     UINT#894,eAxoMessageCategory#Error);
                    DriveStatus.Error.Id := UINT#894;
                    RETURN;
                END_IF;
                IF _retval = WORD#8097 THEN
                    Messenger.Activate(     UINT#895,eAxoMessageCategory#Error);
                    DriveStatus.Error.Id := UINT#895;
                    RETURN;
                END_IF;
                ReadHardwareIOAddress(hardwareID := (AxisRefExt.HWIDs.HW_S_0_0084_0_0) , inputStartAddress => _inputsAddress , inputCount => _inputsCount , outputStartAddress => _outputsAddress , outputCount => _outputsCount);
                IF _inputsCount <> UINT#2 OR _outputsCount <> UINT#0 THEN
                    Messenger.Activate(     UINT#896,eAxoMessageCategory#Error);
                    DriveStatus.Error.Id := UINT#896;
                    RETURN;
                END_IF;
                //************Slot 2 Subslot 8*****************//
                _geoAddr.Subslot:=      UINT#8;
                _geoAddr.Slot   :=      UINT#2;
                _geoAddr.HardwareType := UINT#5; // (5-Submodule)
                _retval := ReadHardwareIDFromSlot(geoAddr := _geoAddr, hardwareID => AxisRefExt.HWIDs.HW_P_0_0106_0_0);
                IF AxisRefExt.HWIDs.HW_P_0_0106_0_0  = UINT#0 THEN
                    Messenger.Activate(     UINT#900,eAxoMessageCategory#Error);
                    DriveStatus.Error.Id := UINT#900;
                    RETURN;
                END_IF;
                IF _retval = WORD#8091 THEN
                    Messenger.Activate(     UINT#901,eAxoMessageCategory#Error);
                    DriveStatus.Error.Id := UINT#901;
                    RETURN;
                END_IF;
                IF _retval = WORD#8094 THEN
                    Messenger.Activate(     UINT#902,eAxoMessageCategory#Error);
                    DriveStatus.Error.Id := UINT#902;
                    RETURN;
                END_IF;
                IF _retval = WORD#8095 THEN
                    Messenger.Activate(     UINT#903,eAxoMessageCategory#Error);
                    DriveStatus.Error.Id := UINT#903;
                    RETURN;
                END_IF;
                IF _retval = WORD#8096 THEN
                    Messenger.Activate(     UINT#904,eAxoMessageCategory#Error);
                    DriveStatus.Error.Id := UINT#904;
                    RETURN;
                END_IF;
                IF _retval = WORD#8097 THEN
                    Messenger.Activate(     UINT#905,eAxoMessageCategory#Error);
                    DriveStatus.Error.Id := UINT#905;
                    RETURN;
                END_IF;
                ReadHardwareIOAddress(hardwareID := (AxisRefExt.HWIDs.HW_P_0_0106_0_0) , inputStartAddress => _inputsAddress , inputCount => _inputsCount , outputStartAddress => _outputsAddress , outputCount => _outputsCount);
                IF _inputsCount <> UINT#2 OR _outputsCount <> UINT#0 THEN
                    Messenger.Activate(     UINT#906,eAxoMessageCategory#Error);
                    DriveStatus.Error.Id := UINT#906;
                    RETURN;
                END_IF;
                //****************************** */
                IF inParent = NULL THEN
                    Messenger.Activate(     UINT#1130,eAxoMessageCategory#Error);
                    DriveStatus.Error.Id := UINT#1130;
                    RETURN;
                END_IF;
                IF AxisRefExt.HWIDs.HW_Device  = UINT#0 THEN
                    Messenger.Activate(     UINT#1131,eAxoMessageCategory#Error);
                    DriveStatus.Error.Id := UINT#1131;
                    RETURN;
                END_IF;
                IF AxisRefExt.HWIDs.HW_Outputs = UINT#0 THEN
                    Messenger.Activate(     UINT#1132,eAxoMessageCategory#Error);
                    DriveStatus.Error.Id := UINT#1132;
                    RETURN;
                END_IF;
                IF AxisRefExt.HWIDs.HW_Inputs = UINT#0 THEN
                    Messenger.Activate(     UINT#1133,eAxoMessageCategory#Error);
                    DriveStatus.Error.Id := UINT#1133;
                    RETURN;
                END_IF;
                IF AxisRefExt.HWIDs.HW_S_0_0134_0_0  = UINT#0 THEN
                    Messenger.Activate(     UINT#1134,eAxoMessageCategory#Error);
                    DriveStatus.Error.Id := UINT#1134;
                    RETURN;
                END_IF;
                IF AxisRefExt.HWIDs.HW_S_0_0145_0_0  = UINT#0 THEN
                    Messenger.Activate(     UINT#1135,eAxoMessageCategory#Error);
                    DriveStatus.Error.Id := UINT#1135;
                    RETURN;
                END_IF;
                IF AxisRefExt.HWIDs.HW_S_0_0282_0_0  = UINT#0 THEN
                    Messenger.Activate(     UINT#1136,eAxoMessageCategory#Error);
                    DriveStatus.Error.Id := UINT#1136;
                    RETURN;
                END_IF;
                IF AxisRefExt.HWIDs.HW_S_0_0259_0_0  = UINT#0 THEN
                    Messenger.Activate(     UINT#1137,eAxoMessageCategory#Error);
                    DriveStatus.Error.Id := UINT#1137;
                    RETURN;
                END_IF;
                IF AxisRefExt.HWIDs.HW_S_0_0260_0_0  = UINT#0 THEN
                    Messenger.Activate(     UINT#1138,eAxoMessageCategory#Error);
                    DriveStatus.Error.Id := UINT#1138;
                    RETURN;
                END_IF;
                IF AxisRefExt.HWIDs.HW_S_0_0359_0_0  = UINT#0 THEN
                    Messenger.Activate(     UINT#1139,eAxoMessageCategory#Error);
                    DriveStatus.Error.Id := UINT#1139;
                    RETURN;
                END_IF;
                IF AxisRefExt.HWIDs.HW_S_0_1720_0_1  = UINT#0 THEN
                    Messenger.Activate(     UINT#1140,eAxoMessageCategory#Error);
                    DriveStatus.Error.Id := UINT#1140;
                    RETURN;
                END_IF;
                IF AxisRefExt.HWIDs.HW_S_0_0092_0_0  = UINT#0 THEN
                    Messenger.Activate(     UINT#1141,eAxoMessageCategory#Error);
                    DriveStatus.Error.Id := UINT#1141;
                    RETURN;
                END_IF;
                IF AxisRefExt.HWIDs.HW_S_0_0080_0_0  = UINT#0 THEN
                    Messenger.Activate(     UINT#1142,eAxoMessageCategory#Error);
                    DriveStatus.Error.Id := UINT#1142;
                    RETURN;
                END_IF;
                IF AxisRefExt.HWIDs.HW_S_0_0193_0_0  = UINT#0 THEN
                    Messenger.Activate(     UINT#1143,eAxoMessageCategory#Error);
                    DriveStatus.Error.Id := UINT#1143;
                    RETURN;
                END_IF;
                IF AxisRefExt.HWIDs.HW_S_0_0135_0_0  = UINT#0 THEN
                    Messenger.Activate(     UINT#1144,eAxoMessageCategory#Error);
                    DriveStatus.Error.Id := UINT#1144;
                    RETURN;
                END_IF;
                IF AxisRefExt.HWIDs.HW_S_0_0144_0_0  = UINT#0 THEN
                    Messenger.Activate(     UINT#1145,eAxoMessageCategory#Error);
                    DriveStatus.Error.Id := UINT#1145;
                    RETURN;
                END_IF;
                IF AxisRefExt.HWIDs.HW_S_0_0386_0_0  = UINT#0 THEN
                    Messenger.Activate(     UINT#1146,eAxoMessageCategory#Error);
                    DriveStatus.Error.Id := UINT#1146;
                    RETURN;
                END_IF;
                IF AxisRefExt.HWIDs.HW_S_0_0535_0_0  = UINT#0 THEN
                    Messenger.Activate(     UINT#1147,eAxoMessageCategory#Error);
                    DriveStatus.Error.Id := UINT#1147;
                    RETURN;
                END_IF;
                IF AxisRefExt.HWIDs.HW_S_0_0390_0_0  = UINT#0 THEN
                    Messenger.Activate(     UINT#1148,eAxoMessageCategory#Error);
                    DriveStatus.Error.Id := UINT#1148;
                    RETURN;
                END_IF;
                IF AxisRefExt.HWIDs.HW_S_0_1720_0_2  = UINT#0 THEN
                    Messenger.Activate(     UINT#1149,eAxoMessageCategory#Error);
                    DriveStatus.Error.Id := UINT#1149;
                    RETURN;
                END_IF;
                IF AxisRefExt.HWIDs.HW_S_0_0084_0_0  = UINT#0 THEN
                    Messenger.Activate(     UINT#1150,eAxoMessageCategory#Error);
                    DriveStatus.Error.Id := UINT#1150;
                    RETURN;
                END_IF;
                IF AxisRefExt.HWIDs.HW_P_0_0106_0_0  = UINT#0 THEN
                    Messenger.Activate(     UINT#1151,eAxoMessageCategory#Error);
                    DriveStatus.Error.Id := UINT#1151;
                    RETURN;
                END_IF;
                _initHwCheckDone    := TRUE;
            END_IF;
            Messenger.ActivateOnCondition(ULINT#1800, NOT _ScalingRead, eAxoMessageCategory#Potential);
            //********************Diagnostics******************//
            HardwareDiagnosticsTask.Run(THIS,AxisRefExt.HWIDs.HW_Device);
            //*******************SCALING***********************//
            IF NOT _ScalingRead THEN
                IF _State = UINT#0 THEN
                    AxisType := eAxoDriveAxisType#Undefined;
                    _State := _State + UINT#1;
                END_IF;
                //Reading Position data scaling: Type (0x2900:01 / S-0-0076 / --) 2byte, binary
                IF _State = UINT#1 THEN                                                                                 //  Scaling type
                    _ReadRecord(    request     :=  TRUE,                                                               //  001: linear scaling:
                                    hardwareID          :=  (AxisRefExt.HWIDs.HW_S_0_0134_0_0),                         //  010: rotary scaling:
                                    index       :=  DINT#76,
                                    maxLength   :=  UINT#2,
                                    record      :=  _data2);
                    Messenger.ActivateOnCondition(ULINT#1801, _ReadRecord.error, eAxoMessageCategory#Error);
                    IF NOT _ReadRecord.busy AND _ReadRecord.valid AND NOT _ReadRecord.error THEN
                        _word.%B0   :=  _data2[0];
                        _word.%B1   :=  _data2[1];
                        _S_0_0076   :=  _word;
                        _State := _State + UINT#1;
                    END_IF;
                END_IF;
                IF _State = UINT#2 THEN                                                                                 //  Scaling type
                    _ReadRecord(request := FALSE, record := _data2);                                                    //  001: linear scaling:
                    IF NOT _ReadRecord.busy AND NOT _ReadRecord.valid AND NOT _ReadRecord.error  THEN                   //  010: rotary scaling:
                        _State :=  _State + UINT#1;
                    END_IF;
                END_IF;
                //Checking the axis type in Position data scaling: Type (0x2900:01 / S-0-0076 / --)
                IF _State = UINT#3 THEN                                                                                 //  Scaling type
                    IF (_S_0_0076 AND WORD#16#0007) = WORD#16#0001 THEN                                                 //  001: linear scaling:
                        AxisType := eAxoDriveAxisType#Linear;                                                           //  010: rotary scaling:
                        _State :=  _State + UINT#1;
                    ELSIF (_S_0_0076 AND WORD#16#0007) = WORD#16#0002 THEN
                        AxisType := eAxoDriveAxisType#Rotary;
                        _State :=  _State + UINT#1;
                    ELSE
                        AxisType := eAxoDriveAxisType#Error;
                        Messenger.ActivateOnCondition(ULINT#1802, TRUE, eAxoMessageCategory#Error);
                        RETURN;
                    END_IF;
                END_IF;
                //Checking the axis unit system in Position data scaling: Type (0x2900:01 / S-0-0076 / --)
                IF _State = UINT#4 THEN                                                                                 //  Unit for linear scaling
                    IF NOT _S_0_0076.%X4 THEN                                                                           //  0: Meter [m]
                        _State :=  _State + UINT#2;                                                                     //  1: Inch [in]
                    ELSE                                                                                                //  Unit for rotary Scaling
                        Messenger.ActivateOnCondition(ULINT#1803, TRUE, eAxoMessageCategory#Error);                     //  0: Angular degree
                        RETURN;                                                                                         //  1: Reserved
                    END_IF;
                END_IF;
                // Irelevant for position, skipping this control.
                // //Checking the axis time base in Position data scaling: Type (0x2900:01 / S-0-0076 / --)
                // IF _State = UINT#5 THEN
                //     IF _S_0_0076.%X5 THEN
                //         _State :=  _State + UINT#1;
                //     ELSE
                //         Messenger.ActivateOnCondition(ULINT#1804, TRUE, eAxoMessageCategory#Error);
                //         RETURN;
                //     END_IF;
                // END_IF;
                //Checking the axis Data reference in Position data scaling: Type (0x2900:01 / S-0-0076 / --)
                IF _State = UINT#6 THEN                                                                                 //  Data reference
                    IF _S_0_0076.%X6 THEN                                                                               //  0: at the motor shaft
                        _State :=  _State + UINT#1;                                                                     //  1: at the load
                    ELSE
                        Messenger.ActivateOnCondition(ULINT#1805, TRUE, eAxoMessageCategory#Error);
                        RETURN;
                    END_IF;
                END_IF;
                //Reading Velocity scaling type (0x2910:01 / S-0-0044 / --) 2byte, binary
                IF _State = UINT#7 THEN                                                                                 //  Scaling type
                    _ReadRecord(    request     :=  TRUE,                                                               //  001: linear scaling:
                                    hardwareID          :=  (AxisRefExt.HWIDs.HW_S_0_0134_0_0),                         //  010: rotary scaling:
                                    index       :=  DINT#44,
                                    maxLength   :=  UINT#2,
                                    record      :=  _data2);
                    Messenger.ActivateOnCondition(ULINT#1806, _ReadRecord.error, eAxoMessageCategory#Error);
                    IF NOT _ReadRecord.busy AND _ReadRecord.valid AND NOT _ReadRecord.error THEN
                        _word.%B0   :=  _data2[0];
                        _word.%B1   :=  _data2[1];
                        _S_0_0044   :=  _word;
                        _State := _State + UINT#1;
                    END_IF;
                END_IF;
                IF _State = UINT#8 THEN                                                                                 //  Scaling type
                    _ReadRecord(request := FALSE, record := _data2);                                                    //  001: linear scaling:
                    IF NOT _ReadRecord.busy AND NOT _ReadRecord.valid AND NOT _ReadRecord.error  THEN                   //  010: rotary scaling:
                        _State :=  _State + UINT#1;
                    END_IF;
                END_IF;
                //Checking the axis type in Velocity scaling type (0x2910:01 / S-0-0044 / --)
                IF _State = UINT#9 THEN                                                                                 //  Scaling type
                    IF (_S_0_0044 AND WORD#16#0007) = WORD#16#0001 AND AxisType = eAxoDriveAxisType#Linear THEN         //  001: linear scaling:
                        _State :=  _State + UINT#1;                                                                     //  010: rotary scaling:
                    ELSIF (_S_0_0044 AND WORD#16#0007) = WORD#16#0002 AND AxisType = eAxoDriveAxisType#Rotary THEN
                        _State :=  _State + UINT#1;
                    ELSE
                        AxisType := eAxoDriveAxisType#Error;
                        Messenger.ActivateOnCondition(ULINT#1807, TRUE, eAxoMessageCategory#Error);
                        RETURN;
                    END_IF;
                END_IF;
                //Checking the axis unit system in Velocity scaling type (0x2910:01 / S-0-0044 / --)
                IF _State = UINT#10 THEN                                                                                //  Unit for linear scaling
                    IF AxisType = eAxoDriveAxisType#Linear AND NOT _S_0_0044.%X4 OR                                     //  0: Millimeter [mm]
                        AxisType = eAxoDriveAxisType#Rotary AND _S_0_0044.%X4 THEN                                      //  1: Inch [in]
                        _State :=  _State + UINT#1;                                                                     //  Unit for rotary scaling
                    ELSE                                                                                                //  0: Revolution
                        Messenger.ActivateOnCondition(ULINT#1808, TRUE, eAxoMessageCategory#Error);                     //  1: Degrees
                        RETURN;
                    END_IF;
                END_IF;
                //Checking the axis time base in Velocity scaling type (0x2910:01 / S-0-0044 / --)
                IF _State = UINT#11 THEN                                                                                //  Unit of time
                    IF _S_0_0044.%X5 THEN                                                                               //  0: Minute [min]
                        _State :=  _State + UINT#1;                                                                     //  1: Second [s]
                    ELSE
                        Messenger.ActivateOnCondition(ULINT#1809, TRUE, eAxoMessageCategory#Error);
                        RETURN;
                    END_IF;
                END_IF;
                //Checking the axis Data reference in Velocity scaling type (0x2910:01 / S-0-0044 / --)
                IF _State = UINT#12 THEN                                                                                //  Data reference
                    IF _S_0_0044.%X6 THEN                                                                               //  0: at the motor shaft
                        _State :=  _State + UINT#1;                                                                     //  1: at the load
                    ELSE
                        Messenger.ActivateOnCondition(ULINT#1810, TRUE, eAxoMessageCategory#Error);
                        RETURN;
                    END_IF;
                END_IF;
                //Reading Acceleration scaling type (0x2920:01 / S-0-0160 / --) 2byte, binary
                IF _State = UINT#13 THEN                                                                                //  Scaling type
                    _ReadRecord(    request     :=  TRUE,                                                               //  001: linear scaling:
                                    hardwareID          :=  (AxisRefExt.HWIDs.HW_S_0_0134_0_0),                         //  010: rotary scaling:
                                    index       :=  DINT#160,                                                           //  011: Ramp time
                                    maxLength   :=  UINT#2,
                                    record      :=  _data2);
                    Messenger.ActivateOnCondition(ULINT#1811, _ReadRecord.error, eAxoMessageCategory#Error);
                    IF NOT _ReadRecord.busy AND _ReadRecord.valid AND NOT _ReadRecord.error THEN
                        _word.%B0   :=  _data2[0];
                        _word.%B1   :=  _data2[1];
                        _S_0_0160   :=  _word;
                        _State := _State + UINT#1;
                    END_IF;
                END_IF;
                IF _State = UINT#14 THEN                                                                                //  Scaling type
                    _ReadRecord(request := FALSE, record := _data2);                                                    //  001: linear scaling:
                    IF NOT _ReadRecord.busy AND NOT _ReadRecord.valid AND NOT _ReadRecord.error  THEN                   //  010: rotary scaling:
                        _State :=  _State + UINT#1;                                                                     //  011: Ramp time
                    END_IF;
                END_IF;
                //Checking the axis type in Acceleration scaling type (0x2920:01 / S-0-0160 / --)
                IF _State = UINT#15 THEN                                                                                //  Scaling type
                    IF (_S_0_0160 AND WORD#16#0007) = WORD#16#0001 AND AxisType = eAxoDriveAxisType#Linear THEN         //  001: linear scaling:
                        _State :=  _State + UINT#1;                                                                     //  010: rotary scaling:
                    ELSIF (_S_0_0160 AND WORD#16#0007) = WORD#16#0002 AND AxisType = eAxoDriveAxisType#Rotary THEN      //  011: Ramp time
                        _State :=  _State + UINT#1;
                    ELSE
                        AxisType := eAxoDriveAxisType#Error;
                        Messenger.ActivateOnCondition(ULINT#1812, TRUE, eAxoMessageCategory#Error);
                        RETURN;
                    END_IF;
                END_IF;
                //Checking the axis unit system in Acceleration scaling type (0x2920:01 / S-0-0160 / --)
                IF _State = UINT#16 THEN                                                                                //  Unit for linear scaling
                    IF NOT _S_0_0160.%X4 THEN                                                                           //  0: Meter [m]
                        _State :=  _State + UINT#1;                                                                     //  1: Inch [in]
                    ELSE                                                                                                //  Unit for rotary scaling
                        Messenger.ActivateOnCondition(ULINT#1813, TRUE, eAxoMessageCategory#Error);                     //  0: Radiant [rad]
                        RETURN;                                                                                         //  1: Reserved
                    END_IF;
                END_IF;
                //Checking the axis time base in Acceleration scaling type (0x2920:01 / S-0-0160 / --)
                IF _State = UINT#17 THEN                                                                                //  Unit of time
                    IF NOT _S_0_0160.%X5 THEN                                                                           //  0: Second [s²]
                        _State :=  _State + UINT#1;                                                                     //  1: Reserved
                    ELSE
                        Messenger.ActivateOnCondition(ULINT#1814, TRUE, eAxoMessageCategory#Error);
                        RETURN;
                    END_IF;
                END_IF;
                //Checking the axis Data reference in Acceleration scaling type (0x2920:01 / S-0-0160 / --)
                IF _State = UINT#18 THEN                                                                                //  Data reference
                    IF _S_0_0160.%X6 THEN                                                                               //  0: at the motor shaft
                        _State :=  _State + UINT#1;                                                                     //  1: at the load
                    ELSE
                        Messenger.ActivateOnCondition(ULINT#1815, TRUE, eAxoMessageCategory#Error);
                        RETURN;
                    END_IF;
                END_IF;
                //Reading Torque/force scaling type (0x2930:01 / S-0-0086 / --) 2byte, binary
                IF _State = UINT#19 THEN                                                                                //  Scaling type
                    _ReadRecord(    request     :=  TRUE,                                                               //  000: Percentage-based scaling (% of reference value)
                                    hardwareID          :=  (AxisRefExt.HWIDs.HW_S_0_0134_0_0),                         //  001: translational scaling (force in N, lbf)
                                    index       :=  DINT#86,                                                            //  010: Rotary scaling (torque in Nm, inlbf)
                                    maxLength   :=  UINT#2,
                                    record      :=  _data2);
                    Messenger.ActivateOnCondition(ULINT#1816, _ReadRecord.error, eAxoMessageCategory#Error);
                    IF NOT _ReadRecord.busy AND _ReadRecord.valid AND NOT _ReadRecord.error THEN
                        _word.%B0   :=  _data2[0];
                        _word.%B1   :=  _data2[1];
                        _S_0_0086   :=  _word;
                        _State := _State + UINT#1;
                    END_IF;
                END_IF;
                IF _State = UINT#20 THEN                                                                                //  Scaling type
                    _ReadRecord(request := FALSE, record := _data2);                                                    //  000: Percentage-based scaling (% of reference value)
                    IF NOT _ReadRecord.busy AND NOT _ReadRecord.valid AND NOT _ReadRecord.error  THEN                   //  001: translational scaling (force in N, lbf)
                        _State :=  _State + UINT#1;                                                                     //  010: Rotary scaling (torque in Nm, inlbf)
                    END_IF;
                END_IF;
                //Checking the axis type in Torque/force scaling type (0x2930:01 / S-0-0086 / --)
                IF _State = UINT#21 THEN                                                                                //  Scaling type
                    IF (_S_0_0086 AND WORD#16#0007) = WORD#16#0001 AND AxisType = eAxoDriveAxisType#Linear THEN         //  000: Percentage-based scaling (% of reference value)
                        _State :=  _State + UINT#1;                                                                     //  001: translational scaling (force in N, lbf)
                    ELSIF (_S_0_0086 AND WORD#16#0007) = WORD#16#0002 AND AxisType = eAxoDriveAxisType#Rotary THEN      //  010: Rotary scaling (torque in Nm, inlbf)
                        _State :=  _State + UINT#1;
                    ELSE
                        AxisType := eAxoDriveAxisType#Error;
                        Messenger.ActivateOnCondition(ULINT#1817, TRUE, eAxoMessageCategory#Error);
                        RETURN;
                    END_IF;
                END_IF;
                //Checking the axis unit system in Torque/force scaling type (0x2930:01 / S-0-0086 / --)
                IF _State = UINT#22 THEN                                                                                //  Unit for force
                    IF NOT _S_0_0086.%X4 THEN                                                                           //  0: newton [N]
                        _State :=  _State + UINT#2;                                                                     //  1: pound-force [lbf]
                    ELSE                                                                                                //  Unit for torque
                        Messenger.ActivateOnCondition(ULINT#1818, TRUE, eAxoMessageCategory#Error);                     //  0: Newton-meter [Nm]
                        RETURN;                                                                                         //  1: inch-pound-force [inlbf]
                    END_IF;
                END_IF;
                // Irelevant for torque, skipping this control.
                // //Checking the axis time base in Torque/force scaling type (0x2930:01 / S-0-0086 / --)
                // IF _State = UINT#23 THEN
                //     IF _S_0_0086.%X5 THEN
                //         _State :=  _State + UINT#1;
                //     ELSE
                //         Messenger.ActivateOnCondition(ULINT#1819, TRUE, eAxoMessageCategory#Error);
                //         RETURN;
                //     END_IF;
                // END_IF;
                //Checking the axis Data reference in Torque/force scaling type (0x2930:01 / S-0-0086 / --)
                IF _State = UINT#24 THEN                                                                                //  Data reference
                    IF _S_0_0086.%X6 THEN                                                                               //  0: at the motor shaft
                        _State :=  _State + UINT#1;                                                                     //  1: at the load
                    ELSE
                        Messenger.ActivateOnCondition(ULINT#1820, TRUE, eAxoMessageCategory#Error);
                        RETURN;
                    END_IF;
                END_IF;
                //Reading Position data scaling: Factor (0x2900:02 / S-0-0077 / --) 2byte, 0 decimal places
                IF _State = UINT#25 THEN
                    _ReadRecord(    request     :=  TRUE,
                                    hardwareID          :=  (AxisRefExt.HWIDs.HW_S_0_0134_0_0),
                                    index       :=  DINT#77,
                                    maxLength   :=  UINT#2,
                                    record      :=  _data2);
                    Messenger.ActivateOnCondition(ULINT#1821, _ReadRecord.error, eAxoMessageCategory#Error);
                    IF NOT _ReadRecord.busy AND _ReadRecord.valid AND NOT _ReadRecord.error THEN
                        _word.%B0   :=  _data2[0];
                        _word.%B1   :=  _data2[1];
                        _S_0_0077   :=  TO_INT(_word);
                        _State := _State + UINT#1;
                    END_IF;
                END_IF;
                IF _State = UINT#26 THEN
                    _ReadRecord(request := FALSE, record := _data2);
                    IF NOT _ReadRecord.busy AND NOT _ReadRecord.valid AND NOT _ReadRecord.error  THEN
                        _State := _State + UINT#1;
                    END_IF;
                END_IF;
                //Reading Position data scaling: Exponent (0x2900:03 / S-0-0078 / --) 2byte, 0 decimal places
                IF _State = UINT#27 THEN
                    _ReadRecord(    request     :=  TRUE,
                                    hardwareID          :=  (AxisRefExt.HWIDs.HW_S_0_0134_0_0),
                                    index       :=  DINT#78,
                                    maxLength   :=  UINT#2,
                                    record      :=  _data2);
                    Messenger.ActivateOnCondition(ULINT#1822, _ReadRecord.error, eAxoMessageCategory#Error);
                    IF NOT _ReadRecord.busy AND _ReadRecord.valid AND NOT _ReadRecord.error THEN
                        _word.%B0   :=  _data2[0];
                        _word.%B1   :=  _data2[1];
                        _S_0_0078   :=  TO_INT(_word);
                        _State := _State + UINT#1;
                    END_IF;
                END_IF;
                IF _State = UINT#28 THEN
                    _ReadRecord(request := FALSE, record := _data2);
                    IF NOT _ReadRecord.busy AND NOT _ReadRecord.valid AND NOT _ReadRecord.error  THEN
                        _State := _State + UINT#1;
                    END_IF;
                END_IF;
                //Reading Rotary position resolution (0x2900:04 / S-0-0079 / --) 4byte, 0 decimal places
                IF _State = UINT#29 THEN
                    _ReadRecord(    request     :=  TRUE,
                                    hardwareID          :=  (AxisRefExt.HWIDs.HW_S_0_0134_0_0),
                                    index       :=  DINT#79,
                                    maxLength   :=  UINT#4,
                                    record      :=  _data4);
                    Messenger.ActivateOnCondition(ULINT#1823, _ReadRecord.error, eAxoMessageCategory#Error);
                    IF NOT _ReadRecord.busy AND _ReadRecord.valid AND NOT _ReadRecord.error THEN
                        _dword.%B0  :=  _data4[0];
                        _dword.%B1  :=  _data4[1];
                        _dword.%B2  :=  _data4[2];
                        _dword.%B3  :=  _data4[3];
                        _S_0_0079   :=  TO_DINT(_dword);
                        _State := _State + UINT#1;
                    END_IF;
                END_IF;
                IF _State = UINT#30 THEN
                    _ReadRecord(request := FALSE, record := _data4);
                    IF NOT _ReadRecord.busy AND NOT _ReadRecord.valid AND NOT _ReadRecord.error  THEN
                        _State := _State + UINT#1;
                    END_IF;
                END_IF;
                //Reading Velocity data scaling: Factor (0x2902:02 / S-0-0045 / --) 2byte, 0 decimal places
                IF _State = UINT#31 THEN
                    _ReadRecord(    request     :=  TRUE,
                                    hardwareID          :=  (AxisRefExt.HWIDs.HW_S_0_0134_0_0),
                                    index       :=  DINT#45,
                                    maxLength   :=  UINT#2,
                                    record      :=  _data2);
                    Messenger.ActivateOnCondition(ULINT#1824, _ReadRecord.error, eAxoMessageCategory#Error);
                    IF NOT _ReadRecord.busy AND _ReadRecord.valid AND NOT _ReadRecord.error THEN
                        _word.%B0   :=  _data2[0];
                        _word.%B1   :=  _data2[1];
                        _S_0_0045   :=  TO_INT(_word);
                        _State := _State + UINT#1;
                    END_IF;
                END_IF;
                IF _State = UINT#32 THEN
                    _ReadRecord(request := FALSE, record := _data2);
                    IF NOT _ReadRecord.busy AND NOT _ReadRecord.valid AND NOT _ReadRecord.error  THEN
                        _State := _State + UINT#1;
                    END_IF;
                END_IF;
                //Reading Velocity data scaling: Exponent (0x2902:03 / S-0-0046 / --) 2byte, 0 decimal places
                IF _State = UINT#33 THEN
                    _ReadRecord(    request     :=  TRUE,
                                    hardwareID          :=  (AxisRefExt.HWIDs.HW_S_0_0134_0_0),
                                    index       :=  DINT#46,
                                    maxLength   :=  UINT#2,
                                    record      :=  _data2);
                    Messenger.ActivateOnCondition(ULINT#1825, _ReadRecord.error, eAxoMessageCategory#Error);
                    IF NOT _ReadRecord.busy AND _ReadRecord.valid AND NOT _ReadRecord.error THEN
                        _word.%B0   :=  _data2[0];
                        _word.%B1   :=  _data2[1];
                        _S_0_0046   :=  TO_INT(_word);
                        _State := _State + UINT#1;
                    END_IF;
                END_IF;
                IF _State = UINT#34 THEN
                    _ReadRecord(request := FALSE, record := _data2);
                    IF NOT _ReadRecord.busy AND NOT _ReadRecord.valid AND NOT _ReadRecord.error  THEN
                        _State := _State + UINT#1;
                    END_IF;
                END_IF;
                //Reading Acceleration data scaling: Factor (0x2904:02 / S-0-0161 / --) 2byte, 0 decimal places
                IF _State = UINT#35 THEN
                    _ReadRecord(    request     :=  TRUE,
                                    hardwareID          :=  (AxisRefExt.HWIDs.HW_S_0_0134_0_0),
                                    index       :=  DINT#161,
                                    maxLength   :=  UINT#2,
                                    record      :=  _data2);
                    Messenger.ActivateOnCondition(ULINT#1826, _ReadRecord.error, eAxoMessageCategory#Error);
                    IF NOT _ReadRecord.busy AND _ReadRecord.valid AND NOT _ReadRecord.error THEN
                        _word.%B0   :=  _data2[0];
                        _word.%B1   :=  _data2[1];
                        _S_0_0161   :=  TO_INT(_word);
                        _State := _State + UINT#1;
                    END_IF;
                END_IF;
                IF _State = UINT#36 THEN
                    _ReadRecord(request := FALSE, record := _data2);
                    IF NOT _ReadRecord.busy AND NOT _ReadRecord.valid AND NOT _ReadRecord.error  THEN
                        _State := _State + UINT#1;
                    END_IF;
                END_IF;
                //Reading Acceleration data scaling: Exponent (0x2904:03 / S-0-0162 / --) 2byte, 0 decimal places
                IF _State = UINT#37 THEN
                    _ReadRecord(    request     :=  TRUE,
                                    hardwareID          :=  (AxisRefExt.HWIDs.HW_S_0_0134_0_0),
                                    index       :=  DINT#162,
                                    maxLength   :=  UINT#2,
                                    record      :=  _data2);
                    Messenger.ActivateOnCondition(ULINT#1827, _ReadRecord.error, eAxoMessageCategory#Error);
                    IF NOT _ReadRecord.busy AND _ReadRecord.valid AND NOT _ReadRecord.error THEN
                        _word.%B0   :=  _data2[0];
                        _word.%B1   :=  _data2[1];
                        _S_0_0162   :=  TO_INT(_word);
                        _State := _State + UINT#1;
                    END_IF;
                END_IF;
                IF _State = UINT#38 THEN
                    _ReadRecord(request := FALSE, record := _data2);
                    IF NOT _ReadRecord.busy AND NOT _ReadRecord.valid AND NOT _ReadRecord.error  THEN
                        _State := _State + UINT#1;
                    END_IF;
                END_IF;
                //Reading Torque/force data scaling: Factor (0x2906:02 / S-0-0093 / --) 2byte, 0 decimal places
                IF _State = UINT#39 THEN
                    _ReadRecord(    request     :=  TRUE,
                                    hardwareID          :=  (AxisRefExt.HWIDs.HW_S_0_0134_0_0),
                                    index       :=  DINT#93,
                                    maxLength   :=  UINT#2,
                                    record      :=  _data2);
                    Messenger.ActivateOnCondition(ULINT#1828, _ReadRecord.error, eAxoMessageCategory#Error);
                    IF NOT _ReadRecord.busy AND _ReadRecord.valid AND NOT _ReadRecord.error THEN
                        _word.%B0   :=  _data2[0];
                        _word.%B1   :=  _data2[1];
                        _S_0_0093   :=  TO_INT(_word);
                        _State := _State + UINT#1;
                    END_IF;
                END_IF;
                IF _State = UINT#40 THEN
                    _ReadRecord(request := FALSE, record := _data2);
                    IF NOT _ReadRecord.busy AND NOT _ReadRecord.valid AND NOT _ReadRecord.error  THEN
                        _State := _State + UINT#1;
                    END_IF;
                END_IF;
                //Reading Torque/force data scaling: Exponent (0x2906:03 / S-0-0094 / --) 2byte, 0 decimal places
                IF _State = UINT#41 THEN
                    _ReadRecord(    request     :=  TRUE,
                                    hardwareID          :=  (AxisRefExt.HWIDs.HW_S_0_0134_0_0),
                                    index       :=  DINT#94,
                                    maxLength   :=  UINT#2,
                                    record      :=  _data2);
                    Messenger.ActivateOnCondition(ULINT#1829, _ReadRecord.error, eAxoMessageCategory#Error);
                    IF NOT _ReadRecord.busy AND _ReadRecord.valid AND NOT _ReadRecord.error THEN
                        _word.%B0   :=  _data2[0];
                        _word.%B1   :=  _data2[1];
                        _S_0_0094   :=  TO_INT(_word);
                        _State := _State + UINT#1;
                    END_IF;
                END_IF;
                IF _State = UINT#42 THEN
                    _ReadRecord(request := FALSE, record := _data2);
                    IF NOT _ReadRecord.busy AND NOT _ReadRecord.valid AND NOT _ReadRecord.error  THEN
                        _State := _State + UINT#1;
                    END_IF;
                END_IF;
                //Reading Inverter type data: Nominal current (0x2314:01 / S-0-0112 / --) 4bytes, 3decimal places
                IF _State = UINT#43 THEN
                    _ReadRecord(    request     :=  TRUE,
                                    hardwareID          :=  (AxisRefExt.HWIDs.HW_S_0_0134_0_0),
                                    index       :=  DINT#112,
                                    maxLength   :=  UINT#4,
                                    record      :=  _data4);
                    Messenger.ActivateOnCondition(ULINT#1830, _ReadRecord.error, eAxoMessageCategory#Error);
                    IF NOT _ReadRecord.busy AND _ReadRecord.valid AND NOT _ReadRecord.error THEN
                        _dword.%B0   :=  _data4[0];
                        _dword.%B1   :=  _data4[1];
                        _dword.%B2   :=  _data4[2];
                        _dword.%B3   :=  _data4[3];
                        _S_0_0112   :=  TO_REAL(TO_INT(_dword)) * REAL#0.001;
                        _State := _State + UINT#1;
                    END_IF;
                END_IF;
                IF _State = UINT#44 THEN
                    _ReadRecord(request := FALSE, record := _data4);
                    IF NOT _ReadRecord.busy AND NOT _ReadRecord.valid AND NOT _ReadRecord.error  THEN
                        _State := _State + UINT#1;
                    END_IF;
                END_IF;
                //Reading Motor torque model: Current constant (0x2018:01 / P-0-0450 / --) 2bytes, 2decimal places
                IF _State = UINT#45 THEN
                    _ReadRecord(    request     :=  TRUE,
                                    hardwareID          :=  (AxisRefExt.HWIDs.HW_S_0_0134_0_0),
                                    index       :=  DINT#4546,
                                    maxLength   :=  UINT#2,
                                    record      :=  _data2);
                    Messenger.ActivateOnCondition(ULINT#1831, _ReadRecord.error, eAxoMessageCategory#Error);
                    IF NOT _ReadRecord.busy AND _ReadRecord.valid AND NOT _ReadRecord.error THEN
                        _word.%B0   :=  _data2[0];
                        _word.%B1   :=  _data2[1];
                        _P_0_0450   :=  TO_REAL(TO_INT(_word)) * REAL#0.01;
                        _State := _State + UINT#1;
                    END_IF;
                END_IF;
                IF _State = UINT#46 THEN
                    _ReadRecord(request := FALSE, record := _data2);
                    IF NOT _ReadRecord.busy AND NOT _ReadRecord.valid AND NOT _ReadRecord.error  THEN
                        _State := _State + UINT#1;
                    END_IF;
                END_IF;
                //Calculating scaling constants
                IF _State = UINT#47 THEN
                    IF AxisType = eAxoDriveAxisType#Linear THEN
                        //  Position
                        ScalingConstantRequiredPosition     :=  _exp[-_S_0_0078 - 3] / TO_LREAL(_S_0_0077);
                        ScalingConstantActualPosition       :=  LREAL#1.0/ScalingConstantRequiredPosition;
                        //  Velocity
                        ScalingConstantRequiredVelocity     :=  _exp[-_S_0_0046 - 3] / TO_LREAL(_S_0_0045);
                        ScalingConstantActualVelocity       :=  LREAL#1.0/ScalingConstantRequiredVelocity;
                        //  Acceleration
                        ScalingConstantRequiredAcceleration :=  _exp[-_S_0_0162 - 3] / TO_LREAL(_S_0_0161);
                        ScalingConstantActualAcceleration   :=  LREAL#1.0/ScalingConstantRequiredAcceleration;
                        //  Deceleration
                        ScalingConstantRequiredDeceleration := ScalingConstantRequiredAcceleration;
                        ScalingConstantActualDeceleration   := ScalingConstantActualAcceleration;
                        //  Torque
                        ScalingConstantActualTorque         := TO_LREAL(_S_0_0093) *_exp[_S_0_0094]; //TO_LREAL(_S_0_0093) *_exp[_S_0_0094 - 2] * TO_LREAL(_P_0_0450) * TO_LREAL(_S_0_0112) ;
                        ScalingConstantRequiredTorque       := LREAL#1.0/ScalingConstantActualTorque;
                        //  Jerk
                        ScalingConstantRequiredJerk         :=  ScalingConstantRequiredAcceleration;
                        ScalingConstantActualJerk           :=  LREAL#1.0/ScalingConstantRequiredJerk;
